FUNCTION_BLOCK E_CALIBRATE (* Event-driven two-point calibration (offset & scale) of an analog input. *)
  (* Standard: 61499-1 *)
  (* Version 2.0, 2026-06-01, Meisterschulen am Ostbahnhof *)
  PACKAGE OSCAT::Basic::POUs::Engineering::measurements;
  (* Documentation:
  Formula
    Y = (X + OFFSET) * SCALE Calibration (Two-Point)
    - Offset (EICO): Apply low reference, set Y_Offset to desired output, fire EICO
   OFFSET := Y_Offset - X → shifts X so that Y = Y_Offset * SCALE at this point
   Note: Only correct when SCALE = 1. See E_CALIBRATE_SQ for a formula that works regardless of SCALE.
   - Scale (EICS): Apply high reference, set Y_Scale to desired output, fire EICS
   SCALE := Y_Scale / (X + OFFSET) → scales so that Y = Y_Scale at this point
    Note: Both Y_Offset and Y_Scale are target values on the output side.
    - REQ (normal operation) is always possible
   - CO must be executed before CS, because CS uses OFFSET
   - This FB does not enforce the order – both EICO and EICS are directly accessible from REQ
   - See E_CALIBRATE_SQ for an ECC-enforced variant
    ECC State Machine
    REQ --EICO--> CO  --1--> REQ     (offset calibration) REQ --EICS--> CS  --1--> REQ     (scale calibration) REQ --REQ---> REQ --1--> REQ     (normal operation) No order enforcement: EICO and EICS are both directly reachable from REQ.
   Key Difference: E_CALIBRATE vs. E_CALIBRATE_SQ
      Feature |  E_CALIBRATE |  E_CALIBRATE_SQ |  
    CO formula |  OFFSET := Y_Offset - X |  OFFSET := Y_Offset / SCALE - X |  
    Y after CO |  Y = Y_Offset * SCALE
   (only correct when SCALE = 1) |  Y = Y_Offset
   (always correct) |  
    Order enforcement |  None (ECC, both accessible from REQ) |  ECC-enforced (CO before CS) |  
     Example
   Scenario: 4–20 mA pressure sensor via logiBUS (0–10 V, normalized to 0.0..1.0).
   Desired output range: 0.0..500.0
      Step |  Action |  Result |  
    1 |  Apply 4 mA (X=0.0), set Y_Offset=0.0, fire EICO |  OFFSET = 0 |  
    2 |  Apply 20 mA (X=1.0), set Y_Scale=500.0, fire EICS |  SCALE = 500 |  
     Output: Y = (X + 0) * 500 = X * 500 = 0..500 ✓
  *)
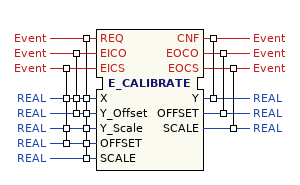
  EVENT_INPUT
    REQ WITH X, Y_Offset, Y_Scale, OFFSET, SCALE; (* Normal Execution Request (berechnet Y) *)
    EICO WITH X, Y_Offset; (* Calibrate Offset (speichert OFFSET := Y_Offset - X) *)
    EICS WITH X, Y_Scale, OFFSET; (* Calibrate Scale (speichert SCALE := Y_Scale / (X + OFFSET)) *)
  END_EVENT
  EVENT_OUTPUT
    CNF WITH Y; (* Execution Confirmed *)
    EOCO WITH OFFSET; (* Offset Calibrated *)
    EOCS WITH SCALE; (* Scale Calibrated *)
  END_EVENT
  VAR_INPUT
    X : REAL; (* Raw input value *)
    Y_Offset : REAL; (* Target output Y at low calibration point (offset) *)
    Y_Scale : REAL; (* Target output Y at high calibration point (scale) *)
  END_VAR
  VAR_OUTPUT
    Y : REAL; (* Calibrated output: Y = (X + OFFSET) * SCALE *)
  END_VAR
  VAR_IN_OUT
    OFFSET : REAL := 0.0; (* Stored offset value *)
    SCALE : REAL := 1.0; (* Stored scale value *)
  END_VAR
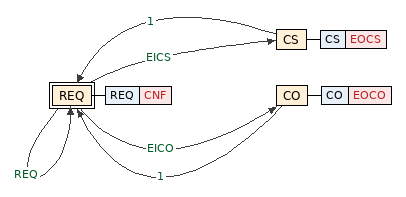
  EC_STATES
    REQ : REQ -> CNF;
    CO : CO -> EOCO;
    CS : CS -> EOCS;
  END_STATES
  EC_TRANSITIONS
    REQ TO CS := EICS;
    REQ TO CO := EICO;
    CS TO REQ := 1;
    CO TO REQ := 1;
    REQ TO REQ := REQ;
  END_TRANSITIONS
  ALGORITHM REQ IN ST:
(* calculate calibrated output *)
Y := (X + OFFSET) * SCALE;
  END_ALGORITHM
  ALGORITHM CO IN ST:
(* store offset so that Y = Y_Offset at current X *)
(* note: after CO, Y = Y_Offset * SCALE, only correct when SCALE = 1 *)
OFFSET := Y_Offset - X;
  END_ALGORITHM
  ALGORITHM CS IN ST:
(* store scale so that Y = Y_Scale at current X (requires OFFSET from CO!) *)
IF (X + OFFSET) <> 0.0 THEN
	SCALE := Y_Scale / (X + OFFSET);
END_IF;
  END_ALGORITHM
END_FUNCTION_BLOCK
